// TIA Portal V18 export
TYPE "UDT_DObasic"
// stored: IsFailsafeCompliant false
   STRUCT
      iID : DInt;   // DOs ID for monitoring
      xInput : Bool;   // Value for DO
      cMOA : Byte;   // Mode Manual/Off/Auto
      xOutput : Bool;   // Phisicl output
      iCounter : Int;   // Counter
      Mark : String["IOmark_string_length"];   // DOs label for monitoring
      xBitCount : Bool;   // Internal
   END_STRUCT;
END_TYPE
